// TIA Portal V20 export
TYPE "mz_LOGSOperationData2"
// stored: Access Published
   STRUCT
      FinReadingQR : Bool;
      DataCatchUp : Bool;
      DataCompareOK : Bool;
      PartClamped : Bool;
      PartUnclamped : Bool;
   END_STRUCT;
END_TYPE
